FUNCTION TFPalletizerGetFormingFromCode : INT
VAR_INPUT
	Forming : POINTER TO ARRAY [1..MAXFORMING] OF TFMachinePalletizer_Forming;
	FCode : INT;
END_VAR
VAR
	pp : INT;
	pf : INT;
	PCode : INT;
END_VAR

(* Per Tutte le Formature Attive *)
FOR pf:=1 TO MAXFORMING DO
	IF Forming^[pf].Enable = 1 THEN
		(* Per tutti i codici di Pallettizzazione *)
		FOR pp:=1 TO MAXFORMINGCODE DO
			IF Forming^[pf].Code[pp] = FCode THEN
				TFPalletizerGetFormingFromCode := pf;
				RETURN;
			END_IF
		END_FOR
	END_IF
END_FOR
TFPalletizerGetFormingFromCode := 0;

END_FUNCTION

(* stored: Version 1.1.0.1, ProductVersion 3.1.4024.11
   POU TFPalletizerGetFormingFromCode: Id {76479c64-953d-4791-a02c-2b610cd7bb02}, SpecialFunc None *)
